(* Bronkhorst mass flow/pressure controller device implementation.
============================================================================================================================================================================================
CONSTRUCTOR TEMPLATE - COPY EVERYTHING BELOW, ADJUST PARAMETERS ACCORDINGLY!
============================================================================================================================================================================================	
(fPredictedFlowCapacity	:= 100, // [REAL] Predicted flow capacity. If logger is provided and the read capacity differs, the error will be reported by the logger.
sPredictedGasType := N2, // [STRING] Predicted gas type. If logger is provided and the read gas type differs, the error will be reported by the logger.
sPredictedFlowUnit := sccm, // [STRING] Predicted flow unit. If logger is provided and the read flow unit differs, the error will be reported by the logger.
iLogger := 0, // [ZigaLibs_Core.I_LoggerEx] Logger implementation provided, set to 0 if not required.
mode := E_ControllerMode.Controlling); // [E_ControllerMode] Controller initial mode
============================================================================================================================================================================================
*)

FUNCTION_BLOCK FB_FlowController EXTENDS ZigaLibs_Core.FB_HasInstanceNameAndPath
VAR_INPUT
	bEnable				: BOOL;	// Enables controller
	fSetpoint			: REAL;	// Setpoint to the controller
	bReadParameters		: BOOL; // Reads CoE parameters on rising edge trigger
END_VAR
VAR_OUTPUT
	fMeassuredValue	: REAL;	// Measured value, reported from the controller
	fValvePosition	: REAL;	// Valve position
END_VAR

// IO
VAR
	Inputs	AT %I*	: ST_ControllerInputs;
	Outputs	AT %Q* 	: ST_ControllerOutputs;
END_VAR

VAR
	bFirstExecution			: BOOL := TRUE;
	_stringBuilder			: ZigaLibs_Core.FB_StringBuilder;
	_CoeList				: ST_ControllerCoeList;
	_logPrefix				: STRING := Tc2_Standard.CONCAT(STR1 := _instancePath, STR2 := ': ');
	_logger					: REFERENCE TO ZigaLibs_Logging.I_Logger;
	_writeLogs				: BOOL;
	_ethercatBoxName		: Tc2_System.T_MaxString;
	{attribute 'hide'} 
	_mode					: E_ControllerMode;	// Hide since mode switching should be logged (done inside the property setter)
	_status					: ST_ControllerStatus;
	_predictedFlowCapacity	: REAL;
	_predictedGasType		: STRING;
	_predictedFlowUnit		: STRING;
	_writeModeRequired					: BOOL;
	_validateModeWrite					: BOOL;
	_controlModeTmp						: E_ControllerMode;
	_coeReadWrite						: ZigaLibs_Core.FB_CoeReadWrite;
	_readParametersRequest				: Tc2_Standard.R_TRIG;
	_parametersReadingInProgress		: BOOL;
	_readBoxName						: ZigaLibs_Core.FB_ReadBoxName;
	_controllerSpeed					: UINT := 1;
	_updateControllerSpeedRequired		: BOOL;
	_validateControllerSpeed			: BOOL;
END_VAR

VAR CONSTANT
	VALVE_FULLY_OPENED_VALUE : REAL := 617.0;
END_VAR

Outputs.ControlByte := BOOL_TO_BYTE(bEnable);

IF bEnable THEN
	Outputs.Setpoint := CalculateSetpointValue();
ELSE
	Outputs.Setpoint := 0;
END_IF

fMeassuredValue := CalculateMeasuredValue();
fValvePosition := 100.0 * UINT_TO_REAL(Inputs.ValvePosition)/VALVE_FULLY_OPENED_VALUE;

IF bFirstExecution THEN
	IF ReadCoE() THEN
		bFirstExecution := FALSE;
	END_IF
END_IF

_readParametersRequest(CLK := bReadParameters);
// Parameters read request
IF _readParametersRequest.Q THEN
	_parametersReadingInProgress := TRUE;
END_IF

IF _parametersReadingInProgress THEN
	IF ReadCoE() THEN
		_parametersReadingInProgress := FALSE;
	END_IF
END_IF

// Controller mode writing and validation
ControllerModeWriting();
// Controller speed writing and validation
ControllerSpeedWriting();

// Status of the controller
_status.ControllerOn := Inputs.StatusWord.0;
_status.SelfOptimization := Inputs.StatusWord.1;
_status.ManualMode := Inputs.StatusWord.2;
_status.SetpointSwitch := Inputs.StatusWord.3;
_status.OptimizationError := Inputs.StatusWord.4;
_status.DataNotValid := Inputs.StatusWord.8;
_status.Overload := Inputs.StatusWord.9;
_status.NetOverload := Inputs.StatusWord.10;

METHOD PRIVATE CalculateMeasuredValue : REAL
VAR_INPUT
END_VAR
CalculateMeasuredValue :=  UINT_TO_REAL(Inputs.MeassuredValue) / LREAL_TO_REAL(EXPT(10,_CoeList.DecimalDigits.Value));
END_METHOD

METHOD PRIVATE CalculateSetpointValue : INT
VAR_INPUT
END_VAR
CalculateSetpointValue := REAL_TO_INT(fSetpoint * LREAL_TO_REAL(EXPT(10, _CoeList.DecimalDigits.Value)));
END_METHOD

{attribute 'monitoring':='call'}
// Gets capacity of the device
PROPERTY Capacity : REAL
GET
Capacity := _CoeList.Capacity.Value;
END_GET
END_PROPERTY

{attribute 'monitoring':='call'}
// Gets the capacity unit of the device
PROPERTY CapacityUnit : STRING(30)
GET
CapacityUnit := _CoeList.CapacityUnit.Value;
END_GET
END_PROPERTY

METHOD PRIVATE ControllerModeWriting
IF _writeModeRequired AND_THEN _coeReadWrite.WriteAny(
		CoeEntry := ADR(_CoeList.ControlMode),
		Value := _mode,
		SlaveAddr := Inputs.AmsAddr)
THEN
	IF _writeLogs THEN
		_logger.LogInfo(message := _stringBuilder.Reset()
			.AddString(str := _logPrefix)
			.AddString(str := 'Finished writing control mode for EtherCAT device ')
			.AddWithDblQuotationMarks(str := _ethercatBoxName)
			.AddString(str := '.')
			.Create());
	END_IF
	_validateModeWrite := TRUE;
	_writeModeRequired := FALSE;
END_IF

IF _validateModeWrite AND_THEN _coeReadWrite.ReadAny(
		CoeEntry := ADR(_CoeList.ControlMode),
		Value := _CoeList.ControlMode.Value,
		SlaveAddr := Inputs.AmsAddr)
THEN
	_validateModeWrite := FALSE;
	IF _writeLogs THEN
		IF _CoeList.ControlMode.Value <> _mode THEN
			// This allows for using TO_STRING on the enum value for better logging experience.
			_controlModeTmp := _CoeList.ControlMode.Value;
			_logger.LogError(message := _stringBuilder.Reset()
				.AddString(str := _logPRefix)
				.AddString('Control mode validation failed! Actual mode read is ')
				.AddWithDblQuotationMarks(str := TO_STRING(_controlModeTmp))
				.AddString(' required mode is ')
				.AddWithDblQuotationMarks(str := TO_STRING(_mode))
				.Create());
		ELSE
			_logger.LogInfo(message := _stringBuilder.Reset()
				.AddString(str := _logPrefix)
				.AddString('Control mode setting validation successful.')
				.Create());
		END_IF
	END_IF
END_IF
END_METHOD

{attribute 'monitoring'='call'}
(*Gets or sets the controller speed.
The controller speed is default set on 1, increasing THIS number will make it faster. 
Please be aware that increasing the controller speed can lead to oscillation when setpoint steps are to steep, 
this will need to be fine-tuned on site to find the optimum setting for the process*)
PROPERTY PUBLIC ControllerSpeed : UINT := 1
GET
ControllerSpeed := _controllerSpeed;
END_GET
SET
IF ControllerSpeed <> _controllerSpeed THEN
	_updateControllerSpeedRequired := TRUE;
END_IF
_controllerSpeed := ControllerSpeed;
END_SET
END_PROPERTY

METHOD PRIVATE ControllerSpeedWriting
VAR_INPUT
END_VAR
IF _updateControllerSpeedRequired AND_THEN _coeReadWrite.WriteAny(
		CoeEntry := ADR(_CoeList.ControllerSpeed),
		Value := _controllerSpeed,
		SlaveAddr := Inputs.AmsAddr)
THEN
	IF _writeLogs THEN
	_logger.LogInfo(message := _stringBuilder.Reset()
		.AddString(str := _logPrefix)
		.AddString(str := 'Finished writing controller speed for EtherCAT device ')
		.AddWithDblQuotationMarks(str := _ethercatBoxName)
		.AddString(str := '.')
		.Create());
	END_IF
	_validateControllerSpeed := TRUE;
	_updateControllerSpeedRequired := FALSE;
END_IF

IF _validateControllerSpeed AND_THEN _coeReadWrite.ReadAny(
		CoeEntry := ADR(_CoeList.ControllerSpeed),
		Value := _CoeList.ControlMode.Value,
		SlaveAddr := Inputs.AmsAddr)
THEN
	_validateControllerSpeed := FALSE;
	IF _writeLogs THEN
		IF _CoeList.ControlMode.Value <> _mode THEN
			_logger.LogError(message := _stringBuilder.Reset()
				.AddString(str := _logPRefix)
				.AddString('Control speed validation failed! Actual speed read is ')
				.AddWithDblQuotationMarks(str := TO_STRING(_CoeList.ControllerSpeed.Value))
				.AddString(' required speed is ')
				.AddWithDblQuotationMarks(str := TO_STRING(_controllerSpeed))
				.Create());
		ELSE
			_logger.LogInfo(message := _stringBuilder.Reset()
				.AddString(str := _logPrefix)
				.AddString('Control speed setting validation successful.')
				.Create());
		END_IF
	END_IF
END_IF
END_METHOD

METHOD FB_init : BOOL
VAR_INPUT
	bInitRetains : BOOL; // if TRUE, the retain variables are initialized (warm start / cold start)
	bInCopyCode : BOOL;  // if TRUE, the instance afterwards gets moved into the copy code (online change)
	
	fPredictedFlowCapacity	: REAL;	// Predicted flow capacity. If bWriteLogs is set to TRUE and the read capacity differs, the error will be reported by the logger.
	sPredictedGasType		: STRING;// Predicted gas type. If bWriteLogs is set to TRUE and the read gas type differs, the error will be reported by the logger.
	sPredictedFlowUnit		: STRING; // Predicted flow unit. If bWriteLogs is set to TRUE and the read flow unit differs, the error will be reported by the logger.
	logger					: REFERENCE TO ZigaLibs_Logging.I_Logger;	// Logger implementation provided, set to 0 if not required.
	mode					: E_ControllerMode;	// Controller initial mode
END_VAR
_predictedFlowCapacity := fPredictedFlowCapacity;
_predictedGasType := sPredictedGasType;
_predictedFlowUnit := sPredictedFlowUnit;
_logger REF= logger;
_mode := mode;
_writeLogs := __ISVALIDREF(logger);
END_METHOD

{attribute 'monitoring':='call'}
// Gets the fluid name of the device
PROPERTY FluidName : STRING(30)
GET
FluidName := _CoeList.FluidName.Value;
END_GET
END_PROPERTY

{attribute 'monitoring':='call'}
// Gets or sets the controller mode
PROPERTY PUBLIC Mode : E_ControllerMode
GET
Mode := _mode;
END_GET
SET
IF _mode <> Mode THEN
	_writeModeRequired := TRUE;
END_IF

_mode := Mode;
END_SET
END_PROPERTY

(* Reads CoE items and updates them. Returns TRUE when done, even if an error occurs. Error is reported to log.*)
METHOD PRIVATE ReadCoE : BOOL
VAR_INST
	eReadCoeStep	: E_ParameterReadingStep;
	bCoeReadError	: BOOL;
	bError			: BOOL;
	fbCoeReadWrite	: ZigaLibs_Core.FB_CoeReadWrite;
END_VAR

VAR CONSTANT
	MAX_REAL_VALUE_DEVIATION : REAL := 0.1;
END_VAR

VAR_INST
	message	: Tc2_System.T_MaxString;
	mfcName	: Tc2_System.T_MaxString;
END_VAR
CASE eReadCoeStep OF
	E_ParameterReadingStep.IDLE:
		ReadCoE := FALSE;
		message := '';
		IF _ethercatBoxName = '' THEN
			_readBoxName(
				AmsNetId := Inputs.AmsAddr,
				PlcRuntimeNetId := '',
				error => bError,
				name => _ethercatBoxName);
		ELSIF _ethercatBoxName <> '' OR bError THEN
			eReadCoeStep := E_ParameterReadingStep.GAS_TYPE;
			IF _writeLogs THEN
				IF NOT bError THEN
					message := _stringBuilder.Reset()	
						.AddString(str := _logPrefix)
						.AddString(str := 'MFC parameters ')
						.AddWithDblQuotationMarks(str := _ethercatBoxName)
						.AddString(str := ':')
						.Create();
				ELSE
					_logger.LogInfo(message := _stringBuilder.Reset()	
						.AddString(str := _logPrefix)
						.AddString(str := 'Reading CoE parameters for Bronkhorst device ')
						.AddWithDblQuotationMarks(str := '<Error reading EC box name>')
						.AddString(str := '...')
						.Create());
				END_IF

			END_IF
		END_IF
		
	E_ParameterReadingStep.GAS_TYPE:
		IF fbCoeReadWrite.ReadAny(
			CoeEntry := ADR(_CoeList.FluidName),
			Value := _CoeList.FluidName.Value,
			SlaveAddr := Inputs.AmsAddr)
		THEN
			_CoeList.FluidName.Value := ZigaLibs_Core.StringHelper.TrimRightSide(_CoeList.FluidName.Value);
			IF _writeLogs THEN
				IF ZigaLibs_Core.StringHelper.TrimRightSide(_CoeList.FluidName.Value) <> _predictedGasType THEN
					_logger.LogWarning(message := _stringBuilder.Reset()
						.AddString(_logPrefix)
						.AddString('Invalid gas type found! Predicted gas type is ')
						.AddWithDblQuotationMarks(_predictedGasType)
						.AddString(' and actual gas type found is ')
						.AddWithDblQuotationMarks(_coeList.FluidName.Value)
						.Create());
				ELSE
					message :=_stringBuilder.Reset()
						.AddString(message)
						.AddString('[')
						.AddString('Gas type: ')
						.AddWithDblQuotationMarks(_coeList.FluidName.Value)
						.AddString(']')
						.Create();
				END_IF
			END_IF
			eReadCoeStep := E_ParameterReadingStep.FLOW_UNIT;
		END_IF
		
	E_ParameterReadingStep.FLOW_UNIT:
		IF fbCoeReadWrite.ReadAny(
			CoeEntry := ADR(_CoeList.CapacityUnit),
			Value := _CoeList.CapacityUnit.Value,
			SlaveAddr := Inputs.AmsAddr)
		THEN
			_CoeList.CapacityUnit.Value := ZigaLibs_Core.StringHelper.TrimRightSide(_CoeList.CapacityUnit.Value);
			IF _writeLogs THEN
				IF ZigaLibs_Core.StringHelper.TrimRightSide(_CoeList.CapacityUnit.Value) <> _predictedFlowUnit THEN
					_logger.LogWarning(message := _stringBuilder.Reset()
						.AddString(_logPrefix)
						.AddString('Invalid flow unit found! Predicted unit is ')
						.AddWithDblQuotationMarks(_predictedFlowUnit)
						.AddString(' and actual flow unit found is ')
						.AddWithDblQuotationMarks(_coeList.CapacityUnit.Value)
						.Create());				
				ELSE
					message :=_stringBuilder.Reset()
						.AddString(message)
						.AddString('[')
						.AddString('Flow unit: ')
						.AddWithDblQuotationMarks(_coeList.CapacityUnit.Value)
						.AddString(']')
						.Create();
				END_IF
			END_IF
			eReadCoeStep := E_ParameterReadingStep.DECIMAL_DIGITS;
		END_IF
		
	E_ParameterReadingStep.DECIMAL_DIGITS:
		IF fbCoeReadWrite.ReadAny(
			CoeEntry := ADR(_CoeList.DecimalDigits),
			Value := _CoeList.DecimalDigits.Value,
			SlaveAddr := Inputs.AmsAddr)
		THEN
			eReadCoeStep := E_ParameterReadingStep.FLOW_CAPACITY;
		END_IF
		
	E_ParameterReadingStep.FLOW_CAPACITY:
		IF fbCoeReadWrite.ReadAny(
			CoeEntry := ADR(_CoeList.Capacity),
			Value := _CoeList.Capacity.Value,
			SlaveAddr := Inputs.AmsAddr)
		THEN
			IF _writeLogs THEN
				IF ABS(_CoeList.Capacity.Value - _predictedFlowCapacity) >= MAX_REAL_VALUE_DEVIATION THEN
					_logger.LogWarning(message := _stringBuilder.Reset()
						.AddString(_logPrefix)
						.AddString('Invalid flow capacity found! Predicted capacity is ')
						.AddString(ZigaLibs_Core.StringConstants.DoubleQuotationMark)
						.AddAnyReal(_predictedFlowCapacity, 3, TRUE).AddString(' ').AddString(_coeList.CapacityUnit.Value)
						.AddString(ZigaLibs_Core.StringConstants.DoubleQuotationMark)
						.AddString(' and actual flow capacity found is ')
						.AddString(ZigaLibs_Core.StringConstants.DoubleQuotationMark)
						.AddAnyReal(_CoeList.Capacity.Value, 3, TRUE).AddString(' ').AddString(_coeList.CapacityUnit.Value)
						.AddString(ZigaLibs_Core.StringConstants.DoubleQuotationMark)
						.AddString('!')
						.Create());
					ELSE
							
					message :=_stringBuilder.Reset()
						.AddString(message)
						.AddString('[')
						.AddString('Flow capacity: ')
						.AddString(ZigaLibs_Core.StringConstants.DoubleQuotationMark)
						.AddAnyReal(_CoeList.Capacity.Value, 3, TRUE).AddString(' ').AddString(_coeList.CapacityUnit.Value)
						.AddString(ZigaLibs_Core.StringConstants.DoubleQuotationMark)
						.AddString(']')
						.Create();
						
					_logger.LogInfo(message);
					END_IF
				END_IF
			eReadCoeStep := E_ParameterReadingStep.IDLE;
			ReadCoE := TRUE;
		END_IF	
END_CASE
END_METHOD

{attribute 'monitoring':='call'}
// Gets the controller status
PROPERTY Status : REFERENCE TO ST_ControllerStatus
GET
Status REF= _status;
END_GET
END_PROPERTY

END_FUNCTION_BLOCK

(* stored: Version 1.1.0.1, ProductVersion 3.1.4024.16
   POU FB_FlowController: Id {4ae6103e-c357-05b9-305d-07911a2f3e97}, SpecialFunc None
   Folder Constructor: Id {1fe8449f-b94f-0219-22c8-3649cc7cb3b5}
   Folder Methods: Id {781a0c72-4665-06e8-0df1-e5645502800d}
   Folder Private: Id {55280652-3923-0ff0-1e6d-a79890bbbafd}
   Folder Properties: Id {fa74778b-e175-0074-22d3-af8310e3452c}
   Folder Public: Id {d42222ef-efab-0798-30b6-38d24b323a35}
   Method CalculateMeasuredValue: Id {ea423dd2-8de1-0f73-3034-64ced1bcd87c}
   Method CalculateSetpointValue: Id {86689ca6-4c77-0658-332d-fdb5f75df13a}
   Property Capacity: Id {151e0e68-21c0-0cd2-1fbe-f6ddb4155f36}
   Get Get: Id {e4917337-5c75-0576-1f6e-fc4f12ed5d88}
   Property CapacityUnit: Id {2b8d7175-dc8f-0228-2ee3-e0fa3fc3423f}
   Get Get: Id {d53e5f36-16a4-0e81-13ff-1ee900c38d84}
   Method ControllerModeWriting: Id {86573b76-921d-091b-05fa-1c781c85c976}
   Property ControllerSpeed: Id {33902a1a-128e-0979-257e-b44f523dabd9}
   Get Get: Id {54a331f5-4c37-0900-0061-fef21ea101f6}
   Set Set: Id {e942ea90-11d2-073e-13fb-7e4be4358ddd}
   Method ControllerSpeedWriting: Id {06283e55-0dfb-0fc5-08c2-23994032f88e}
   Method FB_init: Id {452560b1-3dd5-07ef-1f9c-d7749fdaa339}
   Property FluidName: Id {72233265-6bff-0f7e-33e9-3452c3568c33}
   Get Get: Id {392a6e59-09a9-0957-1857-02c2bbd67f77}
   Property Mode: Id {4c7e1d0e-6e00-01e7-36c0-8b3b117df91e}
   Get Get: Id {e4eff9a5-548f-0608-1fca-54fd16a4d25f}
   Set Set: Id {0d462039-cf9e-0ae0-2cbb-56e6bc7375e2}
   Method ReadCoE: Id {1c46f6b9-c8bc-064d-0797-2b06657f41c3}
   Property Status: Id {0f8f3843-acd8-0cc9-1c5c-b80666ff4a26}
   Get Get: Id {c61a1ec7-9865-0810-09cb-8b3d8a9a65a7} *)
